TYPE Vec13d : ARRAY[1..13] OF LREAL; END_TYPE

(* stored: Version 1.1.0.1, ProductVersion 3.1.4024.12
   DUT Vec13d: Id {67e576c4-46e8-40ba-bc0d-b9106bf65d63} *)
